(* PLC project FiFo Library, CODESYS CODESYS V3.5 SP18 Patch 2, author Toni Kucic *)
(* stored: creationDateTime 2023-02-15T20:34:10.8325937, version 1.0, modificationDateTime 2023-02-15T20:34:07.4157085, organization TK Automation *)
(* Library that holds FIFO and LIFO buffer classes for use in IEC programs *)

TYPE dtFIFO_P_Element_Int : STRUCT
  Value : INT;
  Priority : INT;
END_STRUCT;
END_TYPE

(* Standard FIFO buffer. Allows Enqueing if buffer is not full. After being filled, it has to be emptied completely before further equeueing *)
FUNCTION_BLOCK FIFO_S_INT
  VAR_INPUT
    {attribute 'input_constant'}
    Buffer : POINTER TO INT := 0;  (* Externally allocated buffer. Must be in format ARRAY[0..N]. ! Block doesn't check for Null pointer *)
    {attribute 'input_constant'}
    Size : UINT := 0;  (* Size/Max elements of the buffer *)
  END_VAR
  VAR_OUTPUT
    NrElements : UINT := 0;  (* Number of elements in the FIFO *)
  END_VAR
  VAR
    vHead : INT := -1;  (* Position of the head *)
    vTail : INT := -1;  (* Position of the tail *)
  END_VAR

            
          

(* Returns TRUE if FIFO is empty. Reading not allowed *)
METHOD isEmpty : BOOL
                  isEmpty := vHead = -1 OR vHead > vTail;
RETURN;
                
END_METHOD

(* Returns the next FIFO element stored in the buffer *)
METHOD Dequeue : BOOL
  VAR_OUTPUT
    Value : INT;
  END_VAR
                  IF isEmpty() THEN
    RETURN;
END_IF
Value       := Buffer[vHead];
vHead       := vHead + 1;

NrElements  := NrElements -1;

IF vHead > vTail THEN
    (*Reset*)
    vHead := -1;
    vTail := -1;
    NrElements := 0;
END_IF

Dequeue := TRUE;
RETURN;
                
END_METHOD

(* Inserts new value into the FIFO buffer *)
METHOD Enqueue : BOOL
  VAR_INPUT
    Value : INT;
  END_VAR
                  IF isFull() THEN
    RETURN;
END_IF
IF isEmpty() THEN
    vHead := 0;
END_IF

vTail           := vTail + 1;
Buffer[vTail]   := Value;

NrElements      := NrElements + 1;

Enqueue := TRUE;
RETURN;

                
END_METHOD

(* Returns TRUE if FIFO is full. Inserting not allowed *)
METHOD isFull : BOOL
                  isFull := vTail = Size - 1;
RETURN;
                
END_METHOD

(* Returns the index of the next element to Dequeue. Output paramter holds the element without removing it from the Buffer *)
METHOD Peek : UINT
  VAR_OUTPUT
    Value : INT;
  END_VAR
                  Peek := vHead;
Value:= Buffer[Peek];

RETURN;
                
END_METHOD
END_FUNCTION_BLOCK

(* Circular FIFO buffer. Allows Enqueuing when there is a free space in front of the tail *)
FUNCTION_BLOCK FIFO_C_INT
  VAR_INPUT
    {attribute 'input_constant'}
    Buffer : POINTER TO INT := 0;  (* Externally allocated buffer. Must be in format ARRAY[0..N]. ! Block doesn't check for Null pointer *)
    {attribute 'input_constant'}
    Size : UINT := 0;  (* Size/Max elements of the buffer *)
  END_VAR
  VAR_OUTPUT
    NrElements : UINT := 0;  (* Number of elements in the FIFO *)
  END_VAR
  VAR
    vHead : UINT := 0;  (* Position of the head *)
    vTail : UINT := 0;  (* Position of the tail *)
  END_VAR

            
          

(* Returns the next FIFO element stored in the buffer *)
METHOD Dequeue : BOOL
  VAR_OUTPUT
    Value : INT;
  END_VAR
                  IF isEmpty() THEN
    RETURN;
END_IF

Value       := Buffer[vHead];
vHead       := (vHead + 1) MOD Size;
NrElements  := NrElements - 1;

Dequeue := TRUE;
RETURN;
                
END_METHOD

(* Inserts new value into the FIFO buffer *)
METHOD Enqueue : BOOL
  VAR_INPUT
    Value : INT;
  END_VAR
                  IF isFull() THEN
    RETURN;
END_IF
Buffer[vTail]   := Value;
NrElements      := NrElements + 1;
vTail           := (vTail + 1) MOD Size;

Enqueue := TRUE;
RETURN;
                
END_METHOD

(* Returns TRUE if FIFO is empty. Reading not allowed *)
METHOD isEmpty : BOOL
                  isEmpty := NrElements <= 0;
RETURN;
                
END_METHOD

(* Returns TRUE if FIFO is full. Inserting not allowed *)
METHOD isFull : BOOL
                  isFull := NrElements >= Size;
RETURN;
                
END_METHOD

(* Returns the index of the next element to Dequeue. Output paramter holds the element without removing it from the Buffer *)
METHOD Peek : UINT
  VAR_OUTPUT
    Value : INT;
  END_VAR
                  //Peek := vHead;
//Value:= Buffer[Peek];
Value:= Buffer[Peek := vHead];
RETURN;
                
END_METHOD
END_FUNCTION_BLOCK

(* First word fall trough FIFO buffer. After Dequeuing the whole array is shifted one space to the left so the next element is always at the beggining *)
FUNCTION_BLOCK FIFO_FWFT_INT
  VAR_INPUT
    {attribute 'input_constant'}
    Buffer : POINTER TO INT := 0;  (* Externally allocated buffer. Must be in format ARRAY[0..N]. ! Block doesn't check for Null pointer *)
    {attribute 'input_constant'}
    Size : UINT := 0;  (* Size/Max elements of the buffer *)
  END_VAR
  VAR_OUTPUT
    NrElements : UINT := 0;  (* Number of elements in the FIFO *)
  END_VAR

            
          

(* Returns the next FIFO element stored in the buffer *)
METHOD Dequeue : BOOL
  VAR_OUTPUT
    Value : INT;
  END_VAR
  VAR
    i : UINT;
  END_VAR
                  IF isEmpty() THEN
    RETURN;
END_IF
Value := Buffer[0];

WHILE i < NrElements - 1 DO
    Buffer[i] := Buffer[i+1];
    i := i + 1;
END_WHILE

NrElements := NrElements -1;

Dequeue := TRUE;
RETURN;
                
END_METHOD

(* Inserts new value into the FIFO buffer *)
METHOD Enqueue : BOOL
  VAR_INPUT
    Value : INT;
  END_VAR
                  IF isFull() THEN
    RETURN;
END_IF
Buffer[NrElements] := Value;
NrElements         := NrElements + 1;

Enqueue := TRUE;
RETURN;
                
END_METHOD

(* Returns TRUE if FIFO is empty. Reading not allowed *)
METHOD isEmpty : BOOL
                  isEmpty := NrElements <= 0;
RETURN;
                
END_METHOD

(* Returns TRUE if FIFO is full. Inserting not allowed *)
METHOD isFull : BOOL
                  isFull := NrElements >= Size;
RETURN;
                
END_METHOD

(* Returns the index of the next element to Dequeue. Output paramter holds the element without removing it from the Buffer *)
METHOD Peek : UINT
  VAR_OUTPUT
    Value : INT;
  END_VAR
                  Peek := 0;
Value:= Buffer[Peek];

RETURN;
                
END_METHOD
END_FUNCTION_BLOCK

(* Unordered Priority FIFO buffer. Allows Enqueing if buffer is not full. Dequeues the highest priority elements first. *)
FUNCTION_BLOCK FIFO_UP_INT
  VAR_INPUT
    {attribute 'input_constant'}
    Buffer : POINTER TO dtFIFO_P_Element_Int := 0;  (* Externally allocated buffer. Must be in format ARRAY[0..N]. ! Block doesn't check for Null pointer *)
    {attribute 'input_constant'}
    Size : UINT := 0;  (* Size/Max elements of the buffer *)
  END_VAR
  VAR_OUTPUT
    NrElements : UINT := 0;  (* Number of elements in the FIFO *)
  END_VAR
  VAR
    vLast : INT := -1;  (* Position of the last item *)
  END_VAR

            
          

(* Returns the next FIFO element stored in the buffer *)
METHOD Dequeue : BOOL
  VAR_OUTPUT
    Value : INT;
    Priority : INT;
  END_VAR
  VAR
    vHighestPrioIdx : INT;
    i : INT;
  END_VAR
                  IF isEmpty() THEN
    RETURN;
END_IF

//Get highest priority member
vHighestPrioIdx := Peek();
Value       := Buffer[vHighestPrioIdx].Value;
Priority       := Buffer[vHighestPrioIdx].Priority;

// reduce size of priority queue by first
// shifting all elements one position left
// from index where the highest priority item was found
FOR i := vHighestPrioIdx TO vLast DO
    IF i >= vLast THEN
        EXIT;
    END_IF
    Buffer[i] := Buffer[i+1];
END_FOR
vLast := vLast - 1;

NrElements  := NrElements - 1;

Dequeue := TRUE;
RETURN;
                
END_METHOD

(* Inserts new value into the FIFO buffer *)
METHOD Enqueue : BOOL
  VAR_INPUT
    Value : INT;
    Priority : INT;
  END_VAR
                  IF isFull() THEN
    RETURN;
END_IF
vLast := vLast + 1;

Buffer[vLast].Value         := Value;
Buffer[vLast].Priority      := Priority;
NrElements                  := NrElements + 1;

Enqueue := TRUE;
RETURN;
                
END_METHOD

(* Returns TRUE if FIFO is empty. Reading not allowed *)
METHOD isEmpty : BOOL
                  isEmpty := vLast = -1;
RETURN;
                
END_METHOD

(* Returns TRUE if FIFO is full. Inserting not allowed *)
METHOD isFull : BOOL
                  isFull := vLast = Size - 1;
RETURN;
                
END_METHOD

(* Returns the index of the next element to Dequeue. Output paramter holds the element without removing it from the Buffer *)
METHOD Peek : UINT
  VAR_OUTPUT
    Value : INT;
    Priority : INT;
  END_VAR
  VAR
    maxPrio : INT := -32768;
    i : UINT;
  END_VAR
                  IF isEmpty() THEN
    RETURN;
END_IF

// Linear search for highest priority
FOR i:= 0 TO vLast DO
    // If two items have same priority choose the one with 
    // higher data value 
    IF maxPrio = Buffer[i].Priority AND Buffer[Peek].Value < Buffer[i].Value THEN
        maxPrio := Buffer[i].Priority;
        Peek := i;
        
    // note: using MAX Priority so higher priority number
    // means higher priority
    ELSIF maxPrio < Buffer[i].Priority THEN
        maxPrio := Buffer[i].Priority;
        Peek := i;
    END_IF
END_FOR
Value       := Buffer[Peek].Value;
Priority    := Buffer[Peek].Priority;

RETURN;
                
END_METHOD
END_FUNCTION_BLOCK

(* Ordered Priority FIFO buffer. Allows Enqueing if buffer is not full. Dequeues the highest priority elements first. Buffer is ordered from lowest to highest priority. e.g. 0 = Lowest priority *)
FUNCTION_BLOCK FIFO_OP_INT
  VAR_INPUT
    {attribute 'input_constant'}
    Buffer : POINTER TO dtFIFO_P_Element_Int := 0;  (* Externally allocated buffer. Must be in format ARRAY[0..N]. ! Block doesn't check for Null pointer *)
    {attribute 'input_constant'}
    Size : UINT := 0;  (* Size/Max elements of the buffer *)
  END_VAR
  VAR_OUTPUT
    NrElements : UINT := 0;  (* Number of elements in the FIFO *)
  END_VAR

            
          

(* Returns the next FIFO element stored in the buffer *)
METHOD Dequeue : BOOL
  VAR_OUTPUT
    Value : INT;
    Priority : INT;
  END_VAR
  VAR
    vHighestIdx : INT;
  END_VAR
                  IF isEmpty() THEN
    RETURN;
END_IF

//Get highest priority member
Value       := Buffer[NrElements-1].Value;
Priority    := Buffer[NrElements-1].Priority;

NrElements  := NrElements - 1;

Dequeue := TRUE;
RETURN;
                
END_METHOD

(* Inserts new value into the FIFO buffer *)
METHOD Enqueue : BOOL
  VAR_INPUT
    Value : INT;
    Priority : INT;
  END_VAR
  VAR
    i : INT;
  END_VAR
                  IF isFull() THEN
    RETURN;
END_IF

IF isEmpty() THEN
    Buffer[NrElements].Value         := Value;
    Buffer[NrElements].Priority      := Priority;
    NrElements                       := NrElements + 1;

    Enqueue := TRUE;
    RETURN;
ELSE
    FOR i:= NrElements -1 TO 0 BY -1 DO
        // shift all items rightwards with higher priority
        // than the element we trying to insert
        IF Priority < Buffer[i].Priority THEN
            Buffer[i+1].Value       := Buffer[i].Value;
            Buffer[i+1].Priority    := Buffer[i].Priority;
        ELSE
            EXIT;
        END_IF
    END_FOR
    // insert item just before where
    // lower priority index was found
    Buffer[i+1].Value       := Value;
    Buffer[i+1].Priority    := Priority;
    NrElements              := NrElements + 1;
            
    Enqueue := TRUE;
    RETURN;
END_IF



                
END_METHOD

(* Returns TRUE if FIFO is empty. Reading not allowed *)
METHOD isEmpty : BOOL
                  isEmpty := NrElements = 0;
RETURN;
                
END_METHOD

(* Returns TRUE if FIFO is full. Inserting not allowed *)
METHOD isFull : BOOL
                  isFull := NrElements = Size;
RETURN;
                
END_METHOD

(* Returns the index of the next element to Dequeue. Output paramter holds the element without removing it from the Buffer *)
METHOD Peek : UINT
  VAR_OUTPUT
    Value : INT;
    Priority : INT;
  END_VAR
                  Peek        := NrElements-1;
Value       := Buffer[Peek].Value;
Priority    := Buffer[Peek].Priority;

RETURN;
                
END_METHOD
END_FUNCTION_BLOCK

(* LIFO / Stack buffer. Pushing places new value on top of the stack and poping removes the element from the top. *)
FUNCTION_BLOCK LIFO_INT
  VAR_INPUT
    {attribute 'input_constant'}
    Buffer : POINTER TO INT := 0;  (* Externally allocated buffer. Must be in format ARRAY[0..N]. ! Block doesn't check for Null pointer *)
    {attribute 'input_constant'}
    Size : UINT := 0;  (* Size/Max elements of the buffer *)
  END_VAR
  VAR_OUTPUT
    NrElements : UINT := 0;  (* Number of elements in the FIFO *)
  END_VAR
  VAR
    vTop : INT := -1;  (* Position of the highest element *)
  END_VAR

            
          

(* Returns the top LIFO element stored in the buffer *)
METHOD Pop : BOOL
  VAR_OUTPUT
    Value : INT;
  END_VAR
                  IF isEmpty() THEN
    RETURN;
END_IF

Value       := Buffer[vTop];
vTop        := vTop - 1;
NrElements  := NrElements - 1;

Pop := TRUE;
RETURN;
                
END_METHOD

(* Inserts new value on the top of the LIFO buffer *)
METHOD Push : BOOL
  VAR_INPUT
    Value : INT;
  END_VAR
                  IF isFull() THEN
    RETURN;
END_IF
vTop          := vTop + 1;
Buffer[vTop]  := Value;
NrElements    := NrElements + 1;

Push := TRUE;
RETURN;
                
END_METHOD

(* Returns TRUE if LIFO is empty. Reading not allowed *)
METHOD isEmpty : BOOL
                  isEmpty := vTop = -1;
RETURN;
                
END_METHOD

(* Returns TRUE if LIFO is full. Inserting not allowed *)
METHOD isFull : BOOL
                  isFull := vTop = Size - 1;
RETURN;
                
END_METHOD

(* Returns the index of the next element to Pop. Output paramter holds the element without removing it from the Buffer *)
METHOD Peek : UINT
  VAR_OUTPUT
    Value : INT;
  END_VAR
                  Peek := vTop;
Value:= Buffer[Peek];

RETURN;
                
END_METHOD
END_FUNCTION_BLOCK

PROGRAM FIFO_C_UnitTest
  VAR
    vRunTests : BOOL := FALSE;  (* Tap to TRUE, to run test *)
    vReturnsTrueOnSuccEnqOk : BOOL := FALSE;  (* Results *)
    vFillsThreeValuesOk : BOOL := FALSE;
    vReportsFullOk : BOOL := FALSE;
    vReturnsFalseOnUnSuccEnqOk : BOOL := FALSE;
    vReturnsTrueOnSuccDeqOk : BOOL := FALSE;
    vDequeue1Ok : BOOL := FALSE;
    vDequeue2Ok : BOOL := FALSE;
    vCountingWorks : BOOL := FALSE;
    vReportsEmptyOk : BOOL := FALSE;
    vReturnsTrueOnUnSuccDeqOk : BOOL := FALSE;
    vCirculationOk : BOOL := FALSE;
    vPeekOk : BOOL := FALSE;
    fifo : FIFO_C_INT;
    vFifoBuffer : ARRAY[0..5] OF INT;
    vTempInt : INT;
    vTempIdx : UINT;
  END_VAR

                    (*Init FIFO*)
fifo.FB_Init(bInitRetains := TRUE, bInCopyCode := TRUE); //Implicit function block init, curtesy of codesys. To init function block on every run
SysMemSet(ADR(vFifoBuffer), 0, SIZEOF(vFifoBuffer));
fifo.Buffer := ADR(vFifoBuffer);
fifo.Size   := SIZEOF(vFifoBuffer)/SIZEOF(INT);

(*Test if fifo returns TRUE on successfull enqueue*)
vReturnsTrueOnSuccEnqOk := fifo.Enqueue(1);

(*Test if fifo fills three values correctly*)
fifo.Enqueue(2);
fifo.Enqueue(3);

vFillsThreeValuesOk := vFifoBuffer[0] = 1 AND vFifoBuffer[1] = 2 AND vFifoBuffer[2] = 3;

(*Test if fifo reports FULL when full*)
fifo.Enqueue(4);
fifo.Enqueue(5);
fifo.Enqueue(6);

vReportsFullOk := fifo.isFull();

(*Test if fifo reports FALSE on unsuccesfull enqueue*)
vReturnsFalseOnUnSuccEnqOk := NOT fifo.Enqueue(7);

(*Test if fifo returns TRUE on successfull dequeue*)
vReturnsTrueOnSuccDeqOk := fifo.Dequeue(Value => vTempInt);

(*Test if fifo dequeues values correctly*)
fifo.Dequeue(Value => vTempInt);
vDequeue1Ok := vTempInt = 2;
fifo.Dequeue(Value => vTempInt);
vDequeue2Ok := vTempInt = 3;

(*Test if fifo can count correctly*)
vCountingWorks := fifo.NrElements = 3; //At this point in the tests, there should be 3 elements

(*Test if fifo reports EMPTY when EMPTY*)
fifo.Dequeue(Value => vTempInt); //Returns 4
fifo.Dequeue(Value => vTempInt); //Returns 5
fifo.Dequeue(Value => vTempInt); //Returns 6
vReportsEmptyOk := fifo.isEmpty();

(*Test if fifo reports FALSE on unsuccesfull dequeue*)
vReturnsTrueOnUnSuccDeqOk := NOT fifo.Dequeue();

(*Test if fifo circulates to index 0 after being full and one item dequeued*)
fifo.Enqueue(1);
fifo.Enqueue(2);
fifo.Enqueue(3);
fifo.Enqueue(4);
fifo.Enqueue(5);
fifo.Enqueue(6);
fifo.Dequeue(Value => vTempInt); //Returns 1
fifo.Enqueue(7); //Writes 7 to index 0
vCirculationOk := vFifoBuffer[0] = 7;

(*Test if Peek is ok, should return the next element but not remove it, it should report correct index of the buffer*)
vTempIdx := fifo.Peek(Value => vTempInt);
vPeekOk := fifo.NrElements = 6 AND vTempInt = 2 AND vTempIdx = 1;

vRunTests := FALSE;
                  
END_PROGRAM

PROGRAM FIFO_S_UnitTest
  VAR
    vRunTests : BOOL := FALSE;  (* Tap to TRUE, to run test *)
    vReturnsTrueOnSuccEnqOk : BOOL := FALSE;  (* Results *)
    vFillsThreeValuesOk : BOOL := FALSE;
    vReportsFullOk : BOOL := FALSE;
    vReturnsFalseOnUnSuccEnqOk : BOOL := FALSE;
    vReturnsTrueOnSuccDeqOk : BOOL := FALSE;
    vDequeue1Ok : BOOL := FALSE;
    vDequeue2Ok : BOOL := FALSE;
    vCountingWorks : BOOL := FALSE;
    vReportsEmptyOk : BOOL := FALSE;
    vReturnsTrueOnUnSuccDeqOk : BOOL := FALSE;
    vFifoFullPrevent1Ok : BOOL := FALSE;
    vFifoFullPrevent2Ok : BOOL := FALSE;
    vFifoFullPrevent3Ok : BOOL := FALSE;
    vPeekOk : BOOL := FALSE;
    fifo : FIFO_S_INT;
    vFifoBuffer : ARRAY[0..5] OF INT;
    vTempInt : INT;
    vTempIdx : UINT;
  END_VAR

                    (*Init FIFO*)
fifo.FB_Init(bInitRetains := TRUE, bInCopyCode := TRUE); //Implicit function block init, curtesy of codesys. To init function block on every run
SysMemSet(ADR(vFifoBuffer), 0, SIZEOF(vFifoBuffer));
fifo.Buffer := ADR(vFifoBuffer);
fifo.Size   := SIZEOF(vFifoBuffer)/SIZEOF(INT);

(*Test if fifo returns TRUE on successfull enqueue*)
vReturnsTrueOnSuccEnqOk := fifo.Enqueue(1);

(*Test if fifo fills three values correctly*)
fifo.Enqueue(2);
fifo.Enqueue(3);

vFillsThreeValuesOk := vFifoBuffer[0] = 1 AND vFifoBuffer[1] = 2 AND vFifoBuffer[2] = 3;

(*Test if fifo reports FULL when full*)
fifo.Enqueue(4);
fifo.Enqueue(5);
fifo.Enqueue(6);

vReportsFullOk := fifo.isFull();

(*Test if fifo reports FALSE on unsuccesfull enqueue*)
vReturnsFalseOnUnSuccEnqOk := NOT fifo.Enqueue(7);

(*Test if fifo returns TRUE on successfull dequeue*)
vReturnsTrueOnSuccDeqOk := fifo.Dequeue(Value => vTempInt);

(*Test if fifo dequeues values correctly*)
fifo.Dequeue(Value => vTempInt);
vDequeue1Ok := vTempInt = 2;
fifo.Dequeue(Value => vTempInt);
vDequeue2Ok := vTempInt = 3;

(*Test if fifo can count correctly*)
vCountingWorks := fifo.NrElements = 3; //At this point in the tests, there should be 3 elements

(*Test if fifo reports EMPTY when EMPTY*)
fifo.Dequeue(Value => vTempInt); //Returns 4
fifo.Dequeue(Value => vTempInt); //Returns 5
fifo.Dequeue(Value => vTempInt); //Returns 6
vReportsEmptyOk := fifo.isEmpty();

(*Test if fifo reports FALSE on unsuccesfull dequeue*)
vReturnsTrueOnUnSuccDeqOk := NOT fifo.Dequeue();

(*Test if fifo prevents enqueue if its full*)
fifo.Enqueue(1);
fifo.Enqueue(2);
fifo.Enqueue(3);
fifo.Dequeue(Value => vTempInt); //Returns 1
fifo.Enqueue(4);
fifo.Enqueue(5);
fifo.Enqueue(6); //Here it is full, even though first array index is free
fifo.Enqueue(7); //Writing fails as it is full
vFifoFullPrevent1Ok := fifo.isFull() AND NOT fifo.Enqueue(8);

(*Test if we are able to enqueue again only after empty flag*)
fifo.Dequeue(Value => vTempInt); //4 elems remaining
fifo.Dequeue(Value => vTempInt); //3 elems remaining
fifo.Dequeue(Value => vTempInt); //2 elems remaining
vFifoFullPrevent2Ok := fifo.isFull() AND NOT fifo.Enqueue(8); //Test pass if it still reports full and enqueue fails

fifo.Dequeue(Value => vTempInt); //1 elems remaining
fifo.Dequeue(Value => vTempInt); //0 elems remaining
vFifoFullPrevent3Ok := NOT fifo.isFull() AND fifo.Enqueue(8); //Test pass if it reports empty and enqueue goes trough

(*Test if Peek is ok, should return the next element but not remove it, it should report correct index of the buffer*)
fifo.Enqueue(9);
vTempIdx := fifo.Peek(Value => vTempInt);
vPeekOk := fifo.NrElements = 2 AND vTempInt = 8 AND vTempIdx = 0;

vRunTests := FALSE;
                  
END_PROGRAM

PROGRAM FIFO_FWFT_UnitTest
  VAR
    vRunTests : BOOL := FALSE;  (* Tap to TRUE, to run test *)
    vReturnsTrueOnSuccEnqOk : BOOL := FALSE;  (* Results *)
    vFillsThreeValuesOk : BOOL := FALSE;
    vReportsFullOk : BOOL := FALSE;
    vReturnsFalseOnUnSuccEnqOk : BOOL := FALSE;
    vReturnsTrueOnSuccDeqOk : BOOL := FALSE;
    vDequeue1Ok : BOOL := FALSE;
    vDequeue2Ok : BOOL := FALSE;
    vCountingWorks : BOOL := FALSE;
    vReportsEmptyOk : BOOL := FALSE;
    vReturnsTrueOnUnSuccDeqOk : BOOL := FALSE;
    vFifoFWFTOk : BOOL := FALSE;
    vPeekOk : BOOL := FALSE;
    fifo : FIFO_FWFT_INT;
    vFifoBuffer : ARRAY[0..5] OF INT;
    vTempInt : INT;
    vTempIdx : UINT;
  END_VAR

                    (*Init FIFO*)
fifo.FB_Init(bInitRetains := TRUE, bInCopyCode := TRUE); //Implicit function block init, curtesy of codesys. To init function block on every run
SysMemSet(ADR(vFifoBuffer), 0, SIZEOF(vFifoBuffer));
fifo.Buffer := ADR(vFifoBuffer);
fifo.Size   := SIZEOF(vFifoBuffer)/SIZEOF(INT);

(*Test if fifo returns TRUE on successfull enqueue*)
vReturnsTrueOnSuccEnqOk := fifo.Enqueue(1);

(*Test if fifo fills three values correctly*)
fifo.Enqueue(2);
fifo.Enqueue(3);

vFillsThreeValuesOk := vFifoBuffer[0] = 1 AND vFifoBuffer[1] = 2 AND vFifoBuffer[2] = 3;

(*Test if fifo reports FULL when full*)
fifo.Enqueue(4);
fifo.Enqueue(5);
fifo.Enqueue(6);

vReportsFullOk := fifo.isFull();

(*Test if fifo reports FALSE on unsuccesfull enqueue*)
vReturnsFalseOnUnSuccEnqOk := NOT fifo.Enqueue(7);

(*Test if fifo returns TRUE on successfull dequeue*)
vReturnsTrueOnSuccDeqOk := fifo.Dequeue(Value => vTempInt);

(*Test if fifo dequeues values correctly*)
fifo.Dequeue(Value => vTempInt);
vDequeue1Ok := vTempInt = 2;
fifo.Dequeue(Value => vTempInt);
vDequeue2Ok := vTempInt = 3;

(*Test if fifo can count correctly*)
vCountingWorks := fifo.NrElements = 3; //At this point in the tests, there should be 3 elements

(*Test if fifo reports EMPTY when EMPTY*)
fifo.Dequeue(Value => vTempInt); //Returns 4
fifo.Dequeue(Value => vTempInt); //Returns 5
fifo.Dequeue(Value => vTempInt); //Returns 6
vReportsEmptyOk := fifo.isEmpty();

(*Test if fifo reports FALSE on unsuccesfull dequeue*)
vReturnsTrueOnUnSuccDeqOk := NOT fifo.Dequeue();

(*Test if fifo first word fall trough is working*)
fifo.Enqueue(1);
fifo.Enqueue(2);
fifo.Enqueue(3);
fifo.Dequeue(Value => vTempInt); //Returns 1
fifo.Enqueue(4);
fifo.Enqueue(5);
fifo.Enqueue(6); //Here it is not full, as the first array index is free, compared to Standard fifo, we shifted the whole array to the left, index 0 should hold 2
vFifoFWFTOk := NOT fifo.isFull() AND fifo.Enqueue(7) AND vFifoBuffer[0] = 2;

(*Test if Peek is ok, should return the next element but not remove it, it should report correct index of the buffer*)
vTempIdx := fifo.Peek(Value => vTempInt);
vPeekOk := fifo.NrElements = 6 AND vTempInt = 2 AND vTempIdx = 0;

vRunTests := FALSE;
                  
END_PROGRAM

PROGRAM FIFO_UP_UnitTest
  VAR
    vRunTests : BOOL := FALSE;  (* Tap to TRUE, to run test *)
    vReturnsTrueOnSuccEnqOk : BOOL := FALSE;  (* Results *)
    vFillsThreeValuesOk : BOOL := FALSE;
    vReportsFullOk : BOOL := FALSE;
    vReturnsFalseOnUnSuccEnqOk : BOOL := FALSE;
    vReturnsTrueOnSuccDeqOk : BOOL := FALSE;
    vDequeue1Ok : BOOL := FALSE;
    vDequeue2Ok : BOOL := FALSE;
    vCountingWorks : BOOL := FALSE;
    vReportsEmptyOk : BOOL := FALSE;
    vReturnsTrueOnUnSuccDeqOk : BOOL := FALSE;
    vFifoReturnsHighestPrioValue : BOOL := FALSE;
    vPeekOk : BOOL := FALSE;
    fifo : FIFO_UP_INT;
    vFifoBuffer : ARRAY[0..5] OF dtFIFO_P_Element_Int;
    vTempInt : INT;
    vTempPrio : INT;
    vTempIdx : UINT;
  END_VAR

                    (*Init FIFO*)
fifo.FB_Init(bInitRetains := TRUE, bInCopyCode := TRUE); //Implicit function block init, curtesy of codesys. To init function block on every run
SysMemSet(ADR(vFifoBuffer), 0, SIZEOF(vFifoBuffer));
fifo.Buffer := ADR(vFifoBuffer);
fifo.Size   := SIZEOF(vFifoBuffer)/SIZEOF(dtFIFO_P_Element_Int);

(*Test if fifo returns TRUE on successfull enqueue*)
vReturnsTrueOnSuccEnqOk := fifo.Enqueue(1,1);

(*Test if fifo fills three values correctly*)
fifo.Enqueue(2,2);
fifo.Enqueue(3,3);

vFillsThreeValuesOk := vFifoBuffer[0].Value = 1 AND vFifoBuffer[0].Priority = 1 AND
                       vFifoBuffer[1].Value = 2 AND vFifoBuffer[1].Priority = 2 AND
                       vFifoBuffer[2].Value = 3 AND vFifoBuffer[2].Priority = 3;

(*Test if fifo reports FULL when full*)
fifo.Enqueue(4,4);
fifo.Enqueue(5,5);
fifo.Enqueue(6,6);

vReportsFullOk := fifo.isFull();

(*Test if fifo reports FALSE on unsuccesfull enqueue*)
vReturnsFalseOnUnSuccEnqOk := NOT fifo.Enqueue(7,7);

(*Test if fifo returns TRUE on successfull dequeue*)
vReturnsTrueOnSuccDeqOk := fifo.Dequeue(Value => vTempInt); //Returns 6,6

(*Test if fifo dequeues values correctly*)
fifo.Dequeue(Value => vTempInt, Priority => vTempPrio);
vDequeue1Ok := vTempInt = 5 AND vTempPrio = 5; //Should return the highest priority value, in this case it should be 5,5
fifo.Dequeue(Value => vTempInt, Priority => vTempPrio);
vDequeue2Ok := vTempInt = 4 AND vTempPrio = 4; //Should return the highest priority value, in this case it should be 4,4

(*Test if fifo can count correctly*)
vCountingWorks := fifo.NrElements = 3; //At this point in the tests, there should be 3 elements

(*Test if fifo reports EMPTY when EMPTY*)
fifo.Dequeue(Value => vTempInt, Priority => vTempPrio); //Returns 3,3
fifo.Dequeue(Value => vTempInt, Priority => vTempPrio); //Returns 2,2
fifo.Dequeue(Value => vTempInt, Priority => vTempPrio); //Returns 1,1
vReportsEmptyOk := fifo.isEmpty();

(*Test if fifo reports FALSE on unsuccesfull dequeue*)
vReturnsTrueOnUnSuccDeqOk := NOT fifo.Dequeue();

(*Test if fifo returns the highest priority value first*)
fifo.Enqueue(1,100);
fifo.Enqueue(2,50);
fifo.Enqueue(3,25);
fifo.Enqueue(4,200);
fifo.Enqueue(5,11);
fifo.Enqueue(6,-6);
fifo.Dequeue(Value => vTempInt, Priority => vTempPrio);
vFifoReturnsHighestPrioValue := vTempInt = 4 AND vTempPrio = 200;

(*Test if Peek is ok, should return the next element but not remove it, it should report correct index of the buffer*)
vTempIdx := fifo.Peek(Value => vTempInt, Priority => vTempPrio);
vPeekOk := fifo.NrElements = 5 AND vTempInt = 1 AND vTempIdx = 0;

vRunTests := FALSE;
                  
END_PROGRAM

PROGRAM FIFO_OP_UnitTest
  VAR
    vRunTests : BOOL := FALSE;  (* Tap to TRUE, to run test *)
    vReturnsTrueOnSuccEnqOk : BOOL := FALSE;  (* Results *)
    vFillsThreeValuesOk : BOOL := FALSE;
    vReportsFullOk : BOOL := FALSE;
    vReturnsFalseOnUnSuccEnqOk : BOOL := FALSE;
    vReturnsTrueOnSuccDeqOk : BOOL := FALSE;
    vDequeue1Ok : BOOL := FALSE;
    vDequeue2Ok : BOOL := FALSE;
    vCountingWorks : BOOL := FALSE;
    vReportsEmptyOk : BOOL := FALSE;
    vReturnsTrueOnUnSuccDeqOk : BOOL := FALSE;
    vFifoReturnsHighestPrioValue : BOOL := FALSE;
    vFifoBufferIsOrdered : BOOL := FALSE;
    vPeekOk : BOOL := FALSE;
    fifo : FIFO_OP_INT;
    vFifoBuffer : ARRAY[0..5] OF dtFIFO_P_Element_Int;
    vTempInt : INT;
    vTempPrio : INT;
    vTempIdx : UINT;
  END_VAR

                    (*Init FIFO*)
fifo.FB_Init(bInitRetains := TRUE, bInCopyCode := TRUE); //Implicit function block init, curtesy of codesys. To init function block on every run
SysMemSet(ADR(vFifoBuffer), 0, SIZEOF(vFifoBuffer));
fifo.Buffer := ADR(vFifoBuffer);
fifo.Size   := SIZEOF(vFifoBuffer)/SIZEOF(dtFIFO_P_Element_Int);

(*Test if fifo returns TRUE on successfull enqueue*)
vReturnsTrueOnSuccEnqOk := fifo.Enqueue(1,1);

(*Test if fifo fills three values correctly*)
fifo.Enqueue(2,2);
fifo.Enqueue(3,3);

vFillsThreeValuesOk := vFifoBuffer[0].Value = 1 AND vFifoBuffer[0].Priority = 1 AND
                       vFifoBuffer[1].Value = 2 AND vFifoBuffer[1].Priority = 2 AND
                       vFifoBuffer[2].Value = 3 AND vFifoBuffer[2].Priority = 3;

(*Test if fifo reports FULL when full*)
fifo.Enqueue(4,4);
fifo.Enqueue(5,5);
fifo.Enqueue(6,6);

vReportsFullOk := fifo.isFull();

(*Test if fifo reports FALSE on unsuccesfull enqueue*)
vReturnsFalseOnUnSuccEnqOk := NOT fifo.Enqueue(7,7);

(*Test if fifo returns TRUE on successfull dequeue*)
vReturnsTrueOnSuccDeqOk := fifo.Dequeue(Value => vTempInt); //Returns 6,6

(*Test if fifo dequeues values correctly*)
fifo.Dequeue(Value => vTempInt, Priority => vTempPrio);
vDequeue1Ok := vTempInt = 5 AND vTempPrio = 5; //Should return the highest priority value, in this case it should be 5,5
fifo.Dequeue(Value => vTempInt, Priority => vTempPrio);
vDequeue2Ok := vTempInt = 4 AND vTempPrio = 4; //Should return the highest priority value, in this case it should be 4,4

(*Test if fifo can count correctly*)
vCountingWorks := fifo.NrElements = 3; //At this point in the tests, there should be 3 elements

(*Test if fifo reports EMPTY when EMPTY*)
fifo.Dequeue(Value => vTempInt, Priority => vTempPrio); //Returns 3,3
fifo.Dequeue(Value => vTempInt, Priority => vTempPrio); //Returns 2,2
fifo.Dequeue(Value => vTempInt, Priority => vTempPrio); //Returns 1,1
vReportsEmptyOk := fifo.isEmpty();

(*Test if fifo reports FALSE on unsuccesfull dequeue*)
vReturnsTrueOnUnSuccDeqOk := NOT fifo.Dequeue();

(*Test if fifo returns the highest priority value first*)
fifo.Enqueue(1,100);
fifo.Enqueue(2,50);
fifo.Enqueue(3,25);
fifo.Enqueue(4,200);
fifo.Enqueue(5,11);
fifo.Enqueue(6,-6);
fifo.Dequeue(Value => vTempInt, Priority => vTempPrio);
vFifoReturnsHighestPrioValue := vTempInt = 4 AND vTempPrio = 200;

(*Test if fifo has ordered the buffer correctly according to priority. The buffer is lowest : highest = 0 : N*)
vFifoBufferIsOrdered := vFifoBuffer[0].Value = 6 AND vFifoBuffer[1].Value = 5 AND vFifoBuffer[2].Value = 3 AND vFifoBuffer[3].Value = 2 AND vFifoBuffer[4].Value = 1;

(*Test if Peek is ok, should return the next element but not remove it, it should report correct index of the buffer*)
vTempIdx := fifo.Peek(Value => vTempInt, Priority => vTempPrio);
vPeekOk := fifo.NrElements = 5 AND vTempInt = 1 AND vTempIdx = 4;

vRunTests := FALSE;
                  
END_PROGRAM

PROGRAM LIFO_UnitTest
  VAR
    vRunTests : BOOL := FALSE;  (* Tap to TRUE, to run test *)
    vReturnsTrueOnSuccPushOk : BOOL := FALSE;  (* Results *)
    vFillsThreeValuesOk : BOOL := FALSE;
    vReportsFullOk : BOOL := FALSE;
    vReturnsFalseOnUnSuccPushOk : BOOL := FALSE;
    vReturnsTrueOnSuccPopOk : BOOL := FALSE;
    vPop1Ok : BOOL := FALSE;
    vPop2Ok : BOOL := FALSE;
    vCountingWorks : BOOL := FALSE;
    vReportsEmptyOk : BOOL := FALSE;
    vReturnsTrueOnUnSuccPopOk : BOOL := FALSE;
    vPeekOk : BOOL := FALSE;
    lifo : LIFO_INT;
    vLifoBuffer : ARRAY[0..5] OF INT;
    vTempInt : INT;
    vTempIdx : UINT;
  END_VAR

                    (*Init LIFO*)
lifo.FB_Init(bInitRetains := TRUE, bInCopyCode := TRUE); //Implicit function block init, curtesy of codesys. To init function block on every run
SysMemSet(ADR(vLifoBuffer), 0, SIZEOF(vLifoBuffer));
lifo.Buffer := ADR(vLifoBuffer);
lifo.Size   := SIZEOF(vLifoBuffer)/SIZEOF(INT);

(*Test if lifo returns TRUE on successfull Push*)
vReturnsTrueOnSuccPushOk := lifo.Push(1);

(*Test if lifo fills three values correctly*)
lifo.Push(2);
lifo.Push(3);

vFillsThreeValuesOk := vLifoBuffer[0] = 1 AND vLifoBuffer[1] = 2 AND vLifoBuffer[2] = 3;

(*Test if lifo reports FULL when full*)
lifo.Push(4);
lifo.Push(5);
lifo.Push(6);

vReportsFullOk := lifo.isFull();

(*Test if lifo reports FALSE on unsuccesfull Push*)
vReturnsFalseOnUnSuccPushOk := NOT lifo.Push(7);

(*Test if lifo returns TRUE on successfull Pop*)
vReturnsTrueOnSuccPopOk := lifo.Pop(Value => vTempInt); //Returns 6

(*Test if lifo dequeues values correctly*)
lifo.Pop(Value => vTempInt);
vPop1Ok := vTempInt = 5;
lifo.Pop(Value => vTempInt);
vPop2Ok := vTempInt = 4;

(*Test if lifo can count correctly*)
vCountingWorks := lifo.NrElements = 3; //At this point in the tests, there should be 3 elements

(*Test if lifo reports EMPTY when EMPTY*)
lifo.Pop(Value => vTempInt); //Returns 3
lifo.Pop(Value => vTempInt); //Returns 2
lifo.Pop(Value => vTempInt); //Returns 1
vReportsEmptyOk := lifo.isEmpty();

(*Test if lifo reports FALSE on unsuccesfull Pop*)
vReturnsTrueOnUnSuccPopOk := NOT lifo.Pop();

(*Test if Peek is ok, should return the next element but not remove it, it should report correct index of the buffer*)
lifo.Push(1);
lifo.Push(2);
lifo.Push(3);
vTempIdx := lifo.Peek(Value => vTempInt);
vPeekOk := lifo.NrElements = 3 AND vTempInt = 3 AND vTempIdx = 2;

vRunTests := FALSE;
                  
END_PROGRAM

PROGRAM FIFO_C_ManTest
  VAR
    fifo : FIFO_C_INT;
    fifoa : FIFO_C_INT;
    vFifoBuffer : ARRAY[0..20] OF INT;
    vFifoaBuffer : ARRAY[0..20] OF INT;
    vEnq : BOOL;
    vEnqVal : INT;
    vEnqRet : BOOL;
    vDeq : BOOL;
    vDeqVal : INT;
    vDeqRet : BOOL;
    isFull : BOOL;
    isEmpty : BOOL;
    vCounter : INT;
    vAutoDeq : INT;
  END_VAR

                    (*Initialize the fifos*)
fifo.Buffer := ADR(vFifoBuffer);
fifo.Size   := SIZEOF(vFifoBuffer)/SIZEOF(vFifoBuffer[0]);

fifoa.Buffer := ADR(vFifoaBuffer);
fifoa.Size   := SIZEOF(vFifoaBuffer)/SIZEOF(vFifoaBuffer[0]);

(*Manual testing enqueing and dequeing*)
IF vEnq THEN
    vEnq := FALSE;
    vEnqRet := fifo.Enqueue(vEnqVal);
END_IF

IF vDeq THEN
    vDeq := FALSE;
    vDeqRet := fifo.Dequeue(Value=>vDeqVal);
END_IF
isFull := fifo.isFull();
isEmpty := fifo.isEmpty();
fifo.NrElements;

(*Automatic testing*)
WHILE NOT fifoa.isFull() DO
    vCounter := vCounter + 1;
    fifoa.Enqueue(vCounter);
END_WHILE

IF NOT fifoa.isEmpty() THEN
    fifoa.Dequeue(Value=>vAutoDeq);
END_IF
IF NOT fifoa.isEmpty() THEN
    fifoa.Dequeue(Value=>vAutoDeq);
END_IF
fifoa.NrElements;
                  
END_PROGRAM

PROGRAM FIFO_FWFT_ManTest
  VAR
    fifo : FIFO_FWFT_INT;
    fifoa : FIFO_FWFT_INT;
    vFifoBuffer : ARRAY[0..20] OF INT;
    vFifoaBuffer : ARRAY[0..20] OF INT;
    vEnq : BOOL;
    vEnqVal : INT;
    vEnqRet : BOOL;
    vDeq : BOOL;
    vDeqVal : INT;
    vDeqRet : BOOL;
    isFull : BOOL;
    isEmpty : BOOL;
    vCounter : INT;
    vAutoDeq : INT;
  END_VAR

                    (*Initialize the fifos*)
fifo.Buffer := ADR(vFifoBuffer);
fifo.Size   := SIZEOF(vFifoBuffer)/SIZEOF(vFifoBuffer[0]);

fifoa.Buffer := ADR(vFifoaBuffer);
fifoa.Size   := SIZEOF(vFifoaBuffer)/SIZEOF(vFifoaBuffer[0]);

(*Manual testing enqueing and dequeing*)
IF vEnq THEN
    vEnq := FALSE;
    vEnqRet := fifo.Enqueue(vEnqVal);
END_IF

IF vDeq THEN
    vDeq := FALSE;
    vDeqRet := fifo.Dequeue(Value=>vDeqVal);
END_IF
isFull := fifo.isFull();
isEmpty := fifo.isEmpty();
fifo.NrElements;

(*Automatic testing*)
IF NOT fifoa.isFull() THEN
    vCounter := vCounter + 1;
    fifoa.Enqueue(vCounter);
    fifoa.Enqueue(vCounter+1);
END_IF

IF NOT fifoa.isEmpty() THEN
    fifoa.Dequeue(Value=>vAutoDeq);
END_IF
fifoa.NrElements;

                  
END_PROGRAM

PROGRAM LIFO_ManTest
  VAR
    lifo : LIFO_INT;
    lifoa : LIFO_INT;
    vLifoBuffer : ARRAY[0..20] OF INT;
    vLifoaBuffer : ARRAY[0..20] OF INT;
    vEnq : BOOL;
    vEnqVal : INT;
    vEnqRet : BOOL;
    vDeq : BOOL;
    vDeqVal : INT;
    vDeqRet : BOOL;
    isFull : BOOL;
    isEmpty : BOOL;
    vCounter : INT;
    vAutoDeq : INT;
  END_VAR

                    (*Initialize the fifos*)
lifo.Buffer := ADR(vLifoBuffer);
lifo.Size   := SIZEOF(vLifoBuffer)/SIZEOF(vLifoBuffer[0]);

lifoa.Buffer := ADR(vLifoaBuffer);
lifoa.Size   := SIZEOF(vLifoaBuffer)/SIZEOF(vLifoaBuffer[0]);

(*Manual testing pushing and popping*)
IF vEnq THEN
    vEnq := FALSE;
    vEnqRet := lifo.Push(vEnqVal);
END_IF

IF vDeq THEN
    vDeq := FALSE;
    vDeqRet := lifo.Pop(Value=>vDeqVal);
END_IF
isFull := lifo.isFull();
isEmpty := lifo.isEmpty();
lifo.NrElements;

(*Automatic testing*)
WHILE NOT lifoa.isFull() DO
    vCounter := vCounter + 1;
    lifoa.Push(vCounter);
END_WHILE

IF NOT lifoa.isEmpty() THEN
    lifoa.Pop(Value=>vAutoDeq);
END_IF
lifoa.NrElements;

                  
END_PROGRAM

PROGRAM FIFO_UP_ManTest
  VAR
    fifo : FIFO_UP_INT;
    vFifoBuffer : ARRAY[0..4] OF dtFIFO_P_Element_Int;
    fifoa : FIFO_UP_INT;
    vFifoaBuffer : ARRAY[0..4] OF dtFIFO_P_Element_Int;
    vEnq : BOOL;
    vEnqVal : INT;
    vEnqPrio : INT;
    vEnqRet : BOOL;
    vDeq : BOOL;
    vDeqVal : INT;
    vDeqPrio : INT;
    vDeqRet : BOOL;
    isFull : BOOL;
    isEmpty : BOOL;
    vCounter : INT;
    vAutoDeqValue : INT;
    vAutoDeqPrio : INT;
  END_VAR

                    (*Initialize the fifos*)
fifo.Buffer := ADR(vFifoBuffer);
fifo.Size   := SIZEOF(vFifoBuffer)/SIZEOF(vFifoBuffer[0]);

fifoa.Buffer := ADR(vFifoaBuffer);
fifoa.Size   := SIZEOF(vFifoaBuffer)/SIZEOF(vFifoaBuffer[0]);

(*Manual testing enqueing and dequeing*)
IF vEnq THEN
    vEnq := FALSE;
    vEnqRet := fifo.Enqueue(vEnqVal, vEnqPrio);
END_IF

IF vDeq THEN
    vDeq := FALSE;
    vDeqRet := fifo.Dequeue(Value=>vDeqVal, Priority => vDeqPrio);
END_IF
isFull := fifo.isFull();
isEmpty := fifo.isEmpty();
fifo.NrElements;

(*Automatic testing*)
WHILE NOT fifoa.isFull() DO
    vCounter := vCounter + 1;
    fifoa.Enqueue(Value := vCounter, Priority := vCounter -1);
END_WHILE

IF NOT fifoa.isEmpty() THEN
    fifoa.Dequeue(Value=>vAutoDeqValue, Priority => vAutoDeqPrio);
END_IF
IF NOT fifoa.isEmpty() THEN
    fifoa.Dequeue(Value=>vAutoDeqValue, Priority => vAutoDeqPrio);
END_IF
fifoa.NrElements;
                  
END_PROGRAM

PROGRAM FIFO_S_ManTest
  VAR
    fifo : FIFO_S_INT;
    fifoa : FIFO_S_INT;
    vFifoBuffer : ARRAY[0..20] OF INT;
    vFifoaBuffer : ARRAY[0..20] OF INT;
    vEnq : BOOL;
    vEnqVal : INT;
    vEnqRet : BOOL;
    vDeq : BOOL;
    vDeqVal : INT;
    vDeqRet : BOOL;
    isFull : BOOL;
    isEmpty : BOOL;
    vCounter : INT;
    vAutoDeq : INT;
  END_VAR

                    (*Initialize the fifos*)
fifo.Buffer := ADR(vFifoBuffer);
fifo.Size   := SIZEOF(vFifoBuffer)/SIZEOF(vFifoBuffer[0]);

fifoa.Buffer := ADR(vFifoaBuffer);
fifoa.Size   := SIZEOF(vFifoaBuffer)/SIZEOF(vFifoaBuffer[0]);

(*Manual testing enqueing and dequeing*)
IF vEnq THEN
    vEnq := FALSE;
    vEnqRet := fifo.Enqueue(vEnqVal);
END_IF

IF vDeq THEN
    vDeq := FALSE;
    vDeqRet := fifo.Dequeue(Value=>vDeqVal);
END_IF
isFull := fifo.isFull();
isEmpty := fifo.isEmpty();
fifo.NrElements;

(*Automatic testing*)
WHILE NOT fifoa.isFull() DO
    vCounter := vCounter + 1;
    fifoa.Enqueue(vCounter);
END_WHILE

IF NOT fifoa.isEmpty() THEN
    fifoa.Dequeue(Value=>vAutoDeq);
END_IF
fifoa.NrElements;

                  
END_PROGRAM

PROGRAM FIFO_OP_ManTest
  VAR
    fifo : FIFO_OP_INT;
    vFifoBuffer : ARRAY[0..4] OF dtFIFO_P_Element_Int;
    fifoa : FIFO_OP_INT;
    vFifoaBuffer : ARRAY[0..4] OF dtFIFO_P_Element_Int;
    vEnq : BOOL;
    vEnqVal : INT;
    vEnqPrio : INT;
    vEnqRet : BOOL;
    vDeq : BOOL;
    vDeqVal : INT;
    vDeqPrio : INT;
    vDeqRet : BOOL;
    isFull : BOOL;
    isEmpty : BOOL;
    vCounter : INT;
    vAutoDeqValue : INT;
    vAutoDeqPrio : INT;
  END_VAR

                    (*Initialize the fifos*)
fifo.Buffer := ADR(vFifoBuffer);
fifo.Size   := SIZEOF(vFifoBuffer)/SIZEOF(vFifoBuffer[0]);

fifoa.Buffer := ADR(vFifoaBuffer);
fifoa.Size   := SIZEOF(vFifoaBuffer)/SIZEOF(vFifoaBuffer[0]);

(*Manual testing enqueing and dequeing*)
IF vEnq THEN
    vEnq := FALSE;
    vEnqRet := fifo.Enqueue(vEnqVal, vEnqPrio);
END_IF

IF vDeq THEN
    vDeq := FALSE;
    vDeqRet := fifo.Dequeue(Value=>vDeqVal, Priority => vDeqPrio);
END_IF
isFull := fifo.isFull();
isEmpty := fifo.isEmpty();
fifo.NrElements;

(*Automatic testing*)
WHILE NOT fifoa.isFull() DO
    vCounter := vCounter + 1;
    fifoa.Enqueue(Value := vCounter, Priority := vCounter -1);
END_WHILE

IF NOT fifoa.isEmpty() THEN
    fifoa.Dequeue(Value=>vAutoDeqValue, Priority => vAutoDeqPrio);
END_IF
IF NOT fifoa.isEmpty() THEN
    fifoa.Dequeue(Value=>vAutoDeqValue, Priority => vAutoDeqPrio);
END_IF
fifoa.NrElements;
                  
END_PROGRAM

CONFIGURATION CODESYS_Control_Win_V3_x64
  RESOURCE Application ON PLC
    TASK Task(INTERVAL := T#500ms, PRIORITY := 1);
    TASK FIFO_C_UT_Task(SINGLE := FIFO_C_UnitTest.vRunTests, PRIORITY := 1);
    TASK FIFO_S_UT_Task(SINGLE := FIFO_S_UnitTest.vRunTests, PRIORITY := 1);
    TASK FIFO_FWFT_UT_Task(SINGLE := FIFO_FWFT_UnitTest.vRunTests, PRIORITY := 1);
    TASK FIFO_UP_UT_Task(SINGLE := FIFO_UP_UnitTest.vRunTests, PRIORITY := 1);
    TASK FIFO_OP_UT_Task(SINGLE := FIFO_OP_UnitTest.vRunTests, PRIORITY := 1);
    TASK LIFO_UT_Task(SINGLE := LIFO_UnitTest.vRunTests, PRIORITY := 1);
    PROGRAM FIFO_S_ManTest WITH Task : FIFO_S_ManTest;
    PROGRAM FIFO_FWFT_ManTest WITH Task : FIFO_FWFT_ManTest;
    PROGRAM FIFO_C_ManTest WITH Task : FIFO_C_ManTest;
    PROGRAM FIFO_UP_ManTest WITH Task : FIFO_UP_ManTest;
    PROGRAM LIFO_ManTest WITH Task : LIFO_ManTest;
    PROGRAM FIFO_OP_ManTest WITH Task : FIFO_OP_ManTest;
    PROGRAM FIFO_C_UnitTest WITH FIFO_C_UT_Task : FIFO_C_UnitTest;
    PROGRAM FIFO_S_UnitTest WITH FIFO_S_UT_Task : FIFO_S_UnitTest;
    PROGRAM FIFO_FWFT_UnitTest WITH FIFO_FWFT_UT_Task : FIFO_FWFT_UnitTest;
    PROGRAM FIFO_UP_UnitTest WITH FIFO_UP_UT_Task : FIFO_UP_UnitTest;
    PROGRAM FIFO_OP_UnitTest WITH FIFO_OP_UT_Task : FIFO_OP_UnitTest;
    PROGRAM LIFO_UnitTest WITH LIFO_UT_Task : LIFO_UnitTest;
  END_RESOURCE
END_CONFIGURATION
